// TIA Portal V19 export
TYPE "LubrValve_Wng"
// stored: Access Published
   STRUCT
      SystemNotON : Bool;
   END_STRUCT;
END_TYPE
